// TwinCAT 3 PLC project _03_Command
// ProgramVersion: 3.1.4023.0
// libraries:
//   Tc2_Standard, * (Beckhoff Automation GmbH)
//   Tc2_System, * (Beckhoff Automation GmbH)
//   Tc3_Module, * (Beckhoff Automation GmbH)
// project tree:
//   Command Pattern/Pattern Base/ I_Command.TcIO, NoCommand.TcPOU
//   Command Pattern/ P_Command.TcPOU
//   Command Pattern/Samples/TP10/Clients %28Receivers%29/ Gate.TcPOU (not stored), Light.TcPOU (not stored)
//   Command Pattern/Samples/TP10/Commands/ CloseCommand.TcPOU, I_CloseCommand.TcIO, I_OffCommand.TcIO, I_OnCommand.TcIO, I_OpenCommand.TcIO, OffCommand.TcPOU, OnCommand.TcPOU, OpenCommand.TcPOU
//   Command Pattern/Samples/TP10/Invokers/ Tp10.TcPOU
//   / MAIN.TcPOU, PlcTask.TcTTO
// (motion and I/O tree: see PLC project 13_decorator)
// real-time tasks:
//   TASK PlcTask: cycle T#10ms, priority 20, ADS port 350
// variable links:

CONFIGURATION _03_Command
    RESOURCE PLC ON TwinCAT3
        TASK PlcTask(INTERVAL := T#10ms, PRIORITY := 20);
        PROGRAM MAIN WITH PlcTask : MAIN;
    END_RESOURCE
END_CONFIGURATION

// ---- Command Pattern/Pattern Base/I_Command.TcIO
INTERFACE I_Command

METHOD Execute
VAR_INPUT
END_VAR
END_METHOD

END_INTERFACE

// ---- Command Pattern/Samples/TP10/Commands/I_CloseCommand.TcIO
INTERFACE I_CloseCommand

METHOD Close
END_METHOD

PROPERTY IsClosed : Bool
GET
END_GET
END_PROPERTY

END_INTERFACE

// ---- Command Pattern/Samples/TP10/Commands/I_OffCommand.TcIO
INTERFACE I_OffCommand

PROPERTY IsOff : Bool
GET
END_GET
END_PROPERTY

METHOD Off
END_METHOD

END_INTERFACE

// ---- Command Pattern/Samples/TP10/Commands/I_OnCommand.TcIO
INTERFACE I_OnCommand

PROPERTY IsOn : Bool
GET
END_GET
END_PROPERTY

METHOD On
END_METHOD

END_INTERFACE

// ---- Command Pattern/Samples/TP10/Commands/I_OpenCommand.TcIO
INTERFACE I_OpenCommand

PROPERTY IsOpen : Bool
GET
END_GET
END_PROPERTY

METHOD Open
END_METHOD

END_INTERFACE

// ---- MAIN.TcPOU
PROGRAM MAIN
VAR
END_VAR

(* 
	GOF 		Encapsulate a request as an object, thereby letting you parameterize clients
				with different requests, queue or log requests, and support undoable operations   
*)
P_Command();

END_PROGRAM

// ---- Command Pattern/P_Command.TcPOU
PROGRAM P_Command
VAR
	lightLivingRoom					: Light;
	lightLivingRoomOnCommand		: OnCommand(OnCommand:=LightLivingRoom);
	lightLivingRoomOffCommand		: OffCommand(OffCommand:=LightLivingRoom);

	lightKitchen					: Light;
	lightKitchenOnCommand			: OnCommand(OnCommand:=LightKitchen);
	lightKitchenOffCommand			: OffCommand(OffCommand:=LightKitchen);

	lightBathroom					: Light;
	lightBathroomOnCommand			: OnCommand(OnCommand:=LightBathroom);
	lightBathroomOffCommand			: OffCommand(OffCommand:=LightBathroom);

	frontGate						: Gate;
	frontGateOpenCommand			: OpenCommand(OpenCommand:=frontGate);
	frontGateCloseCommand			: CloseCommand(CloseCommand:=frontGate);
		
	// TP10 (https://fixsus.be/hardware/tp10)
	tp10MainHallway					: TP10;
	
	init							: BOOL := TRUE;// Initialization	
	
END_VAR

IF init THEN
	// assign the commands to the TP10
	tp10MainHallway.SetCommand(0, lightLivingRoomOnCommand);
	tp10MainHallway.SetCommand(5, lightLivingRoomOffCommand);
	tp10MainHallway.SetCommand(1, lightKitchenOnCommand);
	tp10MainHallway.SetCommand(6, lightKitchenOffCommand);
	tp10MainHallway.SetCommand(2, lightBathroomOnCommand);
	tp10MainHallway.SetCommand(7, lightBathroomOffCommand);
	tp10MainHallway.SetCommand(3, frontGateOpenCommand);
	tp10MainHallway.SetCommand(8, frontGateCloseCommand);
	init := FALSE;
END_IF

// The lights have no cyclic call since they just flip the output

// The gate needs to be processed as long as it is not fully opened or closed after a command
frontGate.CyclicCall();

// Process the tp10's, could be an array of instances that is cyclically called
tp10MainHallway.CyclicCall();

END_PROGRAM

// ---- Command Pattern/Samples/TP10/Commands/OnCommand.TcPOU
{attribute 'no_explicit_call' := 'LightOnCommand is a CLASS and must be accessed using methods or properties'}
FUNCTION_BLOCK OnCommand IMPLEMENTS I_Command
VAR
	_onCommand					: I_OnCommand;
END_VAR


// The body of a class must not be used for code.  
// Cyclic code should be called from a method if needed.

METHOD Execute
_onCommand.On();
END_METHOD

METHOD FB_init : BOOL
VAR_INPUT
	bInitRetains : BOOL; // if TRUE, the retain variables are initialized (warm start / cold start)
	bInCopyCode : BOOL;  // if TRUE, the instance afterwards gets moved into the copy code (online change)
	OnCommand			: I_OnCommand;
END_VAR
_onCommand  := OnCommand;
END_METHOD

END_FUNCTION_BLOCK

// ---- Command Pattern/Samples/TP10/Commands/OffCommand.TcPOU
{attribute 'no_explicit_call' := 'LightOnCommand is a CLASS and must be accessed using methods or properties'}
FUNCTION_BLOCK OffCommand IMPLEMENTS I_Command
VAR
	_offCommand					: I_OffCommand;
END_VAR


// The body of a class must not be used for code.  
// Cyclic code should be called from a method if needed.

METHOD Execute
_offCommand.Off();
END_METHOD

METHOD FB_init : BOOL
VAR_INPUT
	bInitRetains : BOOL; // if TRUE, the retain variables are initialized (warm start / cold start)
	bInCopyCode : BOOL;  // if TRUE, the instance afterwards gets moved into the copy code (online change)
	OffCommand			: I_OffCommand;
END_VAR
_offCommand  := OffCommand;
END_METHOD

END_FUNCTION_BLOCK

// ---- Command Pattern/Samples/TP10/Commands/OpenCommand.TcPOU
{attribute 'no_explicit_call' := 'LightOnCommand is a CLASS and must be accessed using methods or properties'}
FUNCTION_BLOCK OpenCommand IMPLEMENTS I_Command
VAR
	_openCommand					: I_OpenCommand;
END_VAR


// The body of a class must not be used for code.  
// Cyclic code should be called from a method if needed.

METHOD Execute
_openCommand.Open();
END_METHOD

METHOD FB_init : BOOL
VAR_INPUT
	bInitRetains : BOOL; // if TRUE, the retain variables are initialized (warm start / cold start)
	bInCopyCode : BOOL;  // if TRUE, the instance afterwards gets moved into the copy code (online change)
	OpenCommand			: I_OpenCommand;
END_VAR
_openCommand  := OpenCommand;
END_METHOD

END_FUNCTION_BLOCK

// ---- Command Pattern/Samples/TP10/Commands/CloseCommand.TcPOU
{attribute 'no_explicit_call' := 'LightOnCommand is a CLASS and must be accessed using methods or properties'}
FUNCTION_BLOCK CloseCommand IMPLEMENTS I_Command
VAR
	_closeCommand					: I_CloseCommand;
END_VAR


// The body of a class must not be used for code.  
// Cyclic code should be called from a method if needed.

METHOD Execute
_closeCommand.Close();
END_METHOD

METHOD FB_init : BOOL
VAR_INPUT
	bInitRetains : BOOL; // if TRUE, the retain variables are initialized (warm start / cold start)
	bInCopyCode : BOOL;  // if TRUE, the instance afterwards gets moved into the copy code (online change)
	CloseCommand			: I_CloseCommand;
END_VAR
_closeCommand  := CloseCommand;
END_METHOD

END_FUNCTION_BLOCK

// ---- Command Pattern/Samples/TP10/Invokers/Tp10.TcPOU
{attribute 'no_explicit_call' := 'Tp10 is a CLASS and must be accessed using methods or properties'}
FUNCTION_BLOCK Tp10
VAR
	buttons			AT%I*		: ARRAY[0..NOOFCOMMANDS-1] OF BOOL;
	risingTrigger				: ARRAY[0..NOOFCOMMANDS-1] OF R_TRIG;

	commands					: ARRAY[0..NOOFCOMMANDS-1] OF I_Command;
	noCommand					: NoCommand;	// Default command containing NO code in Execute
END_VAR
VAR CONSTANT
	NOOFCOMMANDS				: INT := 10;
END_VAR
/// https://fixsus.be/hardware/tp10


// The body of a class must not be used for code.  
// Cyclic code should be called from a method if needed.

METHOD CyclicCall

VAR
	i: INT;
END_VAR
// Check the pushbuttons
FOR i := 0 TO NOOFCOMMANDS -1 DO
	risingTrigger[i](CLK:=buttons[i]);
	// Issue command if the button was pressed
	IF risingTrigger[i].Q		THEN
		commands[i].Execute();		
	END_IF
END_FOR
END_METHOD

METHOD FB_init : BOOL
VAR_INPUT
	bInitRetains : BOOL; // if TRUE, the retain variables are initialized (warm start / cold start)
	bInCopyCode : BOOL;  // if TRUE, the instance afterwards gets moved into the copy code (online change)
END_VAR
VAR
	i					: INT;
END_VAR
// Initialize the command buttons to NOCommand 
FOR i := 0 TO NOOFCOMMANDS - 1 DO
	Commands[i] := THIS^.noCommand;		// basic initialization of a button, avoids the need of checking for a valid command in the code, just does nothing when pressed
END_FOR
END_METHOD

METHOD RemoveCommand
VAR_INPUT
	slot					: INT;
END_VAR
// Check if the slot no is valid
IF slot >=0 AND slot < NOOFCOMMANDS THEN 
	commands[slot] := noCommand;	
END_IF
END_METHOD

METHOD SetCommand
VAR_INPUT
	slot					: INT;
	command					: I_Command;
END_VAR
// Check if the slot no is valid
IF slot >=0 AND slot < NOOFCOMMANDS THEN 
	commands[slot] := command;	
END_IF
END_METHOD

END_FUNCTION_BLOCK

// ---- Command Pattern/Pattern Base/NoCommand.TcPOU
{attribute 'no_explicit_call' := 'NoCommand is a CLASS and must be accessed using methods or properties'}
FUNCTION_BLOCK NoCommand IMPLEMENTS I_Command
VAR
END_VAR
/// Command that does nothing for base initialization

METHOD Execute
END_METHOD

END_FUNCTION_BLOCK
